(* CODESYS project Trabalho_final.project

Project tree, tasks and I/O mapping:
  Device : CODESYS Control Win V3, 3S - Smart Software Solutions GmbH, order no. 305021, version 3.5.11.40
    application Application
      libraries: Standard, * (System)
      task MainTask (cyclic, interval t#20ms, priority 1) calls Mode_Selection, Sequencia_Processo, Resetar, C_Automatico, Quantidade_Gin, Quantidade_Vermouth, Quantidade_tanque01, Quantidade_refrigerante, Temperatura, Quantidade_tanque02, c_resetar_tanque01, Sistema_esteira, C_Automatico_Tonel
      global variables GVL
      program Quantidade_Gin [ST]
      program Quantidade_Vermouth [ST]
      program Quantidade_refrigerante [ST]
      program Quantidade_tanque01 [ST]
      program Temperatura [ST]
      program C_Automatico [SFC]: Step3_active, Step7_active, Liga_motor_Abre_refrigerante_active, Resetar_active, Step3_active_0, Step2_active, Step4_active, Step5_active, Step6_active, Step7_active_0, Step8_active, Step10_active, Step9_active, Step12_active
      program Quantidade_tanque02 [ST]
      program Sistema_esteira [ST]
      program Mode_Selection [LD]
      program Resetar [ST]
      program Sequencia_Processo [SFC]: Step4_active, Automatico_active
      program c_resetar_tanque01 [ST]
      program C_Automatico_Tonel [SFC]: Step0_active, Step1_active, Step2_active, Step1_active_0
      program C_EMG [ST]
*)

// Device/Application/GVL
{attribute 'qualified_only'}
VAR_GLOBAL
	Mensagem : STRING[255] := 'NADA AINDA';
	
	//Modos de execução 
	Liga							  : BOOL;
	Sistema_ativo					  : BOOL;
	Selecao							  : BOOL := FALSE;  // 0 para automatico, 1 para o remoto
	Selecionado						  : BOOL;
	EMG								  : BOOL;	// Sistema de emergencia 
	Modo_manual 					  : BOOL;	// Indica que esta em modo manual
	Modo_automatico					  : BOOL;	// Indica que esta em modo automatico
	
	// controles do sistema 
	resetar : BOOL := FALSE;
	ativador_automatico	: BOOL := FALSE;
	resetar_tanque01 : BOOL := FALSE;
	
	// Colocar 30 litros de gin 
	Valvula_gin                       : BOOL := FALSE;   // Atuador válvula de gin
	Quantidade_gin					  : REAL := 0.0;     // Quantidade de gin (L)
	Temporizador_gin				  : TON; 			// De atuação 7,5S
	
	//Colocar 15 litros de vermouth 
	Valvula_vermouth                  : BOOL := FALSE;   // Válvula de vermouth
	Quantidade_vermouth			      : REAL := 0.0;     // Quantidade de vermouth (L)
	Temporizador_vermouth			  : TON;				// De atuação 4.5s 
	
	// Colocar Líquido Refrigerante
	Valvula_liquido_refrigerante      : BOOL := FALSE;   // Entrada de líquido refrigerante
	Quantidade_liquido_refrigerante	  : REAL := 0.0;     // Quantidade de liquido refrigerante (L)
	Valvula_descarte_refrigerante     : BOOL := FALSE;   // Válvula de descarte do refrigerante
    Alto_nivel_refrigerante           : BOOL := FALSE;   // Nível alto refrigerante
    Baixo_nivel_refrigerante          : BOOL := FALSE;   // Nível baixo refrigerante
	Temporizador_entrada_refrigerante : TON;
	Temporizador_saida_refrigerante : TON;
	
	// Tanque 01 quantidades 
	Tanque01_vazio                    : BOOL := TRUE;   // Sensor tanque 1 vazio
	Quantidade_liquido                : REAL := 0.0;     // Quantidade do líquido (L)
	Tanque01_30L                      : BOOL := FALSE;   // Sensor tanque(30L)
	Tanque01_45L                      : BOOL := FALSE;   // Sensor tanque(45L)
	Tanque01_50L                      : BOOL := FALSE;   // Sensor tanque(50L)
	Temporizador_produto			  : TON;
	Temporizador_produto_T2			  : TON;
	
	// Temperaturas
	Ativador_temperatura :BOOL:=FALSE;
 	Temporizador_temperatura		 : TON;
    Termometro_produto_0C            : BOOL := FALSE;   // Sensor que indica que a temperatura esta 0°c
	Temperatura_produto            	 : REAL := 27.0;     // Temperatura do produto
	
	//Bloco 01
	Motor_tanque01                   : BOOL := FALSE;   // Motor do tanque 01
	
	//Bloco de ligamento 
    Valvula_envio_produto            : BOOL := FALSE;   // Envio do produto
    Bomba_entre_tanques              : BOOL := FALSE;   // Bomba de transferência
    Valvula_rejeitos                 : BOOL := FALSE;   // Válvula para rejeitos
    Valvula_envio_tanque02           : BOOL := FALSE;   // Válvula de envio ao tanque 02
    
	//Bloco 02
	Tanque02_190l                    : BOOL := FALSE;   // Sensor tanque 2 cheio (190L)
	Quantidade_liquido_02            : REAL := 0.0;     // Quantidade do líquido em bloco 02 (L)
    Tanque02_95_por100               : BOOL := FALSE;   // Tanque 2 a 95% => 188,005 => 188L
    Tanque02_85_por100               : BOOL := FALSE;   // Tanque 2 a 85% => 168,215 => 168L
	Tanque02_50_por100               : BOOL := FALSE;   // Tanque 2 a 50% => 98,95 => 98L
    Tanque02_10_por100               : BOOL := FALSE;   // Tanque 2 a 10% => 19,79L  => 19L
	Temporizador_saida_tonel : TON;
	
	CarregamentoCompleto : BOOL:=FALSE;
	
	Timer_Inicia_Esvaziamento : TON;   // 5 segundos
    Timer_Retira_Produto : TON;       // 0.5 segundos
    Timer_Finaliza_Esgotamento : TON; // 3 segundos
	
	
	
	// Quantidade tonel 
    Valvula_produto_tonel            : BOOL := FALSE;   // Válvula para o tonel final
	Quantidade_liquido_tonel         : REAL := 0.0;     // Quantidade do líquido no tonel (L)
	Tonel_cheio                      : BOOL := FALSE;   // tonel cheio
	Tonel_pretaparado 				 : BOOL := FALSE;	// Sensor que indica que o tonel esta na boca da valvula
	Temporizador_produ_tonel		 : TON; 
	
	//Quantidade de toneis 
	Quantidade_tonel_produzido       : REAL := 0.0;     // Quantidade de toneis produzida
	Quantidade_tonel_liberada        : REAL := 0.0;     // Quantidade de toneis liberadas
	
	// esteira
    Esteira_tonel                    : BOOL := FALSE;   // Esteira transportadora
	Sensor_tonel 					 :BOOL := FALSE;
END_VAR

// Device/Application/Mode_Selection
PROGRAM Mode_Selection
VAR
END_VAR

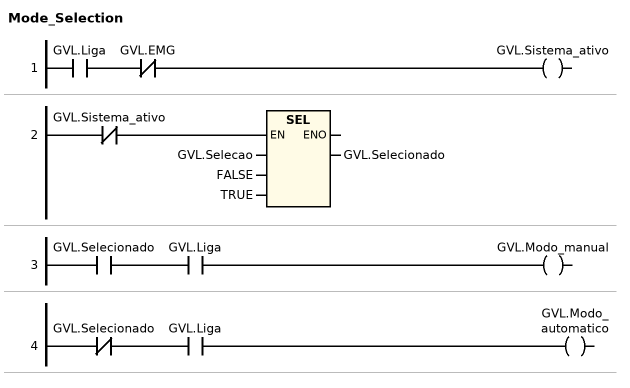
// NETWORK 1
GVL.Sistema_ativo := GVL.Liga AND NOT GVL.EMG;

// NETWORK 2
IF NOT GVL.Sistema_ativo THEN GVL.Selecionado := SEL(GVL.Selecao, FALSE, TRUE); END_IF

// NETWORK 3
GVL.Modo_manual := GVL.Selecionado AND GVL.Liga;

// NETWORK 4
GVL.Modo_automatico := NOT GVL.Selecionado AND GVL.Liga;

END_PROGRAM

// Device/Application/Sequencia_Processo
PROGRAM Sequencia_Processo
VAR
END_VAR

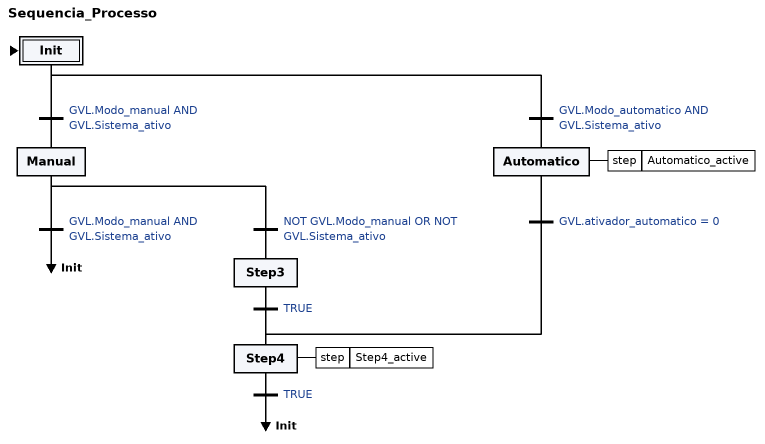
INITIAL_STEP Init:
END_STEP
TRANSITION FROM Init TO Manual
    := GVL.Modo_manual AND GVL.Sistema_ativo;
END_TRANSITION
STEP Manual:
END_STEP
TRANSITION FROM Manual TO Init
    := GVL.Modo_manual AND GVL.Sistema_ativo;
END_TRANSITION
TRANSITION FROM Manual TO Step3
    := NOT GVL.Modo_manual OR NOT GVL.Sistema_ativo;
END_TRANSITION
STEP Step3:
END_STEP
TRANSITION FROM Step3 TO Step4
    := TRUE;
END_TRANSITION
TRANSITION FROM Init TO Automatico
    := GVL.Modo_automatico AND GVL.Sistema_ativo;
END_TRANSITION
STEP Automatico:
    Automatico_active(N);  // step action
END_STEP
TRANSITION FROM Automatico TO Step4
    := GVL.ativador_automatico = 0;
END_TRANSITION
STEP Step4:
    Step4_active(N);  // step action
END_STEP
TRANSITION FROM Step4 TO Init
    := TRUE;
END_TRANSITION

ACTION Step4_active:
IF GVL.resetar = 0 THEN
	GVL.resetar := 1;
END_IF
END_ACTION

ACTION Automatico_active:
IF GVL.ativador_automatico = 0 THEN
	GVL.ativador_automatico := 1;
END_IF
END_ACTION

END_PROGRAM

// Device/Application/Resetar
PROGRAM Resetar
VAR
END_VAR


IF GVL.resetar = 1 THEN
	GVL.Valvula_gin                 			:= FALSE;
	GVL.Quantidade_gin              			:= 0.0;
	GVL.Valvula_vermouth            			:= FALSE;
	GVL.Quantidade_vermouth         			:= 0.0;
	GVL.Valvula_liquido_refrigerante 			:= FALSE;
	GVL.Quantidade_liquido_refrigerante			:= 0.0;
	GVL.Valvula_descarte_refrigerante 			:= FALSE;
	GVL.Alto_nivel_refrigerante      			:= FALSE;
	GVL.Baixo_nivel_refrigerante     			:= TRUE;
	GVL.Tanque01_vazio              			:= TRUE;
	GVL.Quantidade_liquido          			:= 0.0;
	GVL.Tanque01_30L                			:= FALSE;
	GVL.Tanque01_45L                			:= FALSE;
	GVL.Tanque01_50L                			:= FALSE;
	GVL.Termometro_produto_0C       			:= FALSE;
	GVL.Temperatura_produto         			:= 27.0;
	GVL.Motor_tanque01              			:= FALSE;
	GVL.Valvula_envio_produto       			:= FALSE;
	GVL.Bomba_entre_tanques         			:= FALSE;
	GVL.Valvula_rejeitos            			:= FALSE;
	GVL.Valvula_envio_tanque02      			:= FALSE;
	GVL.Tanque02_190l               			:= FALSE;
	GVL.Quantidade_liquido_02       			:= 0.0;
	GVL.Tanque02_95_por100          			:= FALSE;
	GVL.Tanque02_85_por100          			:= FALSE;
	GVL.Tanque02_50_por100          			:= FALSE;
	GVL.Tanque02_10_por100          			:= FALSE;
	GVL.Valvula_produto_tonel       			:= FALSE;
	GVL.Quantidade_liquido_tonel    			:= 0.0;
	GVL.Tonel_cheio                 			:= FALSE;
	GVL.Tonel_pretaparado           			:= FALSE;
	GVL.Quantidade_tonel_produzido  			:= 0.0;
	GVL.Quantidade_tonel_liberada   			:= 0.0;
	GVL.Esteira_tonel               			:= FALSE;
	GVL.resetar 								:= FALSE;
END_IF

END_PROGRAM

// Device/Application/Quantidade_Gin
PROGRAM Quantidade_Gin
VAR
	Limite_gin : REAL;
END_VAR

// ====================================================
//            CONTROLE DA VALVULA DE GIN
// ====================================================


// --------------------------------------
// Definição do limite por modo
// --------------------------------------
IF (GVL.Modo_manual = 1) THEN
    Limite_gin := 52;   // Modo Manual
ELSIF (GVL.Modo_automatico = 1) THEN
    Limite_gin := 30;   // Modo Automático
END_IF


// --------------------------------------
// Condições gerais de operação
// --------------------------------------
IF (GVL.EMG = 0) THEN

    // --------------------------------------
    // Se válvula está aberta
    // --------------------------------------
    IF GVL.Valvula_gin = 1 THEN

        // Fecha válvula quando atingir limite
        IF GVL.Quantidade_gin >= Limite_gin THEN
            GVL.Valvula_gin := 0;
        ELSE
            // Liga temporizador para contar 0.5 s
            GVL.Temporizador_gin(IN := TRUE, PT := T#0.5S);

            // Quando temporizador finalizar, incrementa volume
            IF GVL.Temporizador_gin.Q THEN

                //  equivalente a 4 L/s → 2 L a cada 0.5s
                GVL.Quantidade_gin      := GVL.Quantidade_gin + 2;
                GVL.Quantidade_liquido  := GVL.Quantidade_liquido + 2;

                // Reseta TON para permitir novo ciclo de 0.5s
                GVL.Temporizador_gin(IN := FALSE);
            END_IF

        END_IF

    ELSE
        // Válvula fechada → garantimos TON desligado
        GVL.Temporizador_gin(IN := FALSE);
    END_IF

ELSE
    // Se emergência ativa → TON off
    GVL.Temporizador_gin(IN := FALSE);
END_IF

END_PROGRAM

// Device/Application/Quantidade_Vermouth
PROGRAM Quantidade_Vermouth 
VAR
	Limite_vermouth : REAL;
END_VAR

// ====================================================
//        CONTROLE DA VÁLVULA DE VERMOUTH
// ====================================================


// --------------------------------------
// Definição do limite por modo
// --------------------------------------
IF (GVL.Modo_manual = 1) THEN
    Limite_vermouth := 51;    // Modo Manual → limite do líquido total
ELSIF (GVL.Modo_automatico = 1) THEN
    Limite_vermouth := 14;    // Modo Automático → limite específico do vermouth
END_IF



// --------------------------------------
// Condições gerais de operação
// --------------------------------------
IF (GVL.EMG = 0) THEN

    // --------------------------------------
    // Se a válvula está aberta
    // --------------------------------------
    IF GVL.Valvula_vermouth = 1 THEN

        // Fecha válvula quando atingir limite
        IF GVL.Quantidade_vermouth >= Limite_vermouth THEN

            GVL.Valvula_vermouth := 0;

            // Ajustes específicos do automático
            IF (GVL.Modo_automatico = 1) THEN
                GVL.Quantidade_liquido  := 45;
                GVL.Quantidade_vermouth := 15;
            END_IF

        ELSE
            // Liga temporizador para contar 0.5 s
            GVL.Temporizador_vermouth(IN := TRUE, PT := T#0.5S);

            // Quando temporizador finalizar, incrementa volume
            IF GVL.Temporizador_vermouth.Q THEN

                // Vazão: 3,33 L/s → 1,665 L a cada 0.5 s
                GVL.Quantidade_vermouth := GVL.Quantidade_vermouth + 1.665;
                GVL.Quantidade_liquido  := GVL.Quantidade_liquido  + 1.665;

                // Reseta TON para novo ciclo
                GVL.Temporizador_vermouth(IN := FALSE);
            END_IF

        END_IF

    ELSE
        // Válvula fechada → garante TON desligado
        GVL.Temporizador_vermouth(IN := FALSE);
    END_IF


ELSE
    // Se emergência ativa → TON desligado
    GVL.Temporizador_vermouth(IN := FALSE);
END_IF

END_PROGRAM

// Device/Application/C_Automatico
PROGRAM C_Automatico
VAR
END_VAR

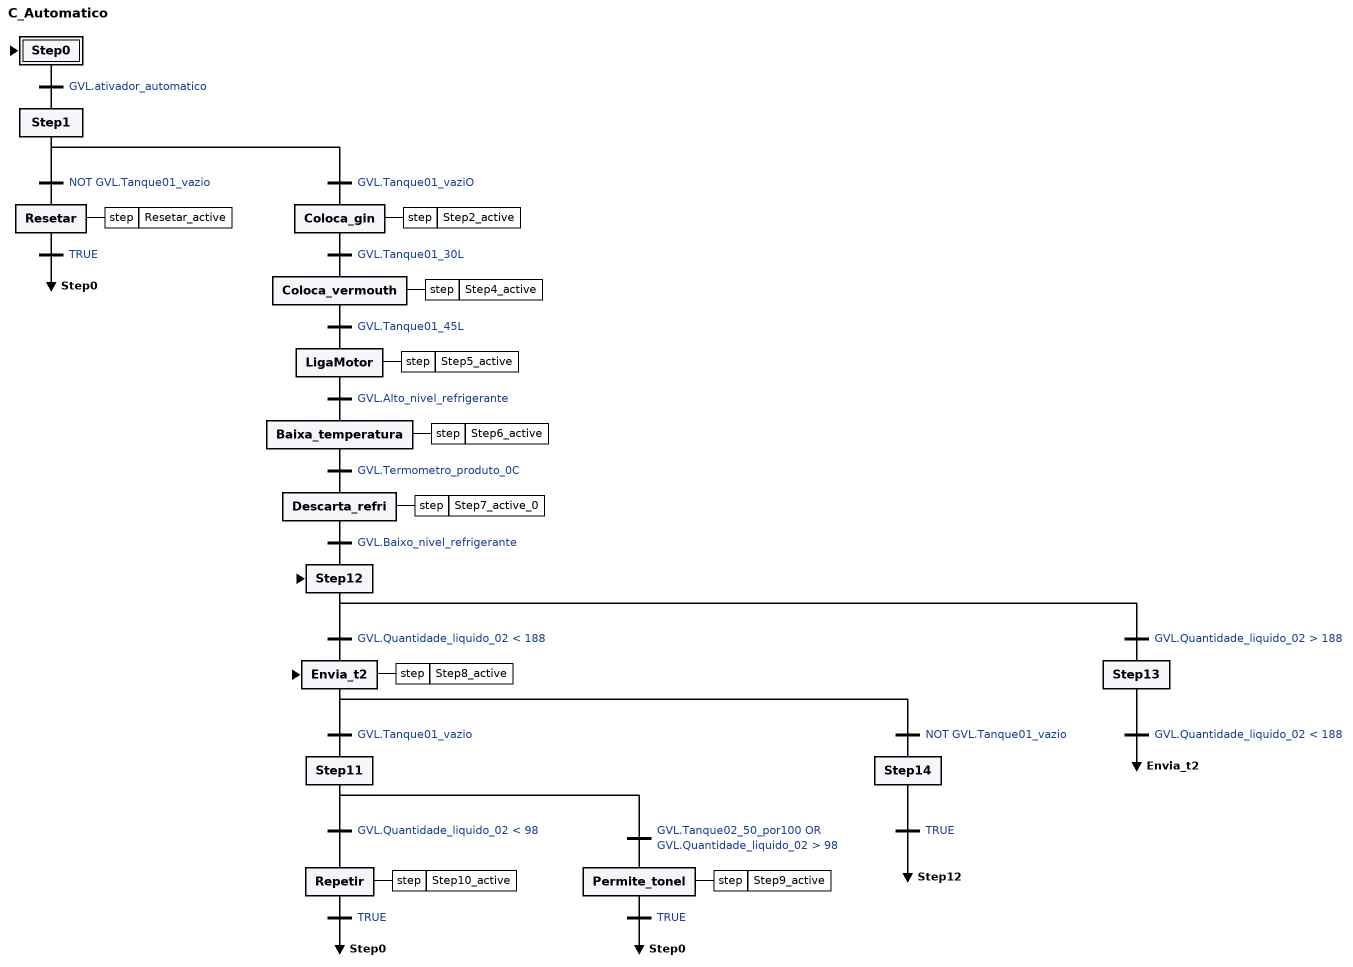
INITIAL_STEP Step0:
END_STEP
TRANSITION FROM Step0 TO Step1
    := GVL.ativador_automatico;
END_TRANSITION
STEP Step1:
END_STEP
TRANSITION FROM Step1 TO Resetar
    := NOT GVL.Tanque01_vazio;
END_TRANSITION
STEP Resetar:
    Resetar_active(N);  // step action
END_STEP
TRANSITION FROM Resetar TO Step0
    := TRUE;
END_TRANSITION
TRANSITION FROM Step1 TO Coloca_gin
    := GVL.Tanque01_vaziO;
END_TRANSITION
STEP Coloca_gin:
    Step2_active(N);  // step action
END_STEP
TRANSITION FROM Coloca_gin TO Coloca_vermouth
    := GVL.Tanque01_30L;
END_TRANSITION
STEP Coloca_vermouth:
    Step4_active(N);  // step action
END_STEP
TRANSITION FROM Coloca_vermouth TO LigaMotor
    := GVL.Tanque01_45L;
END_TRANSITION
STEP LigaMotor:
    Step5_active(N);  // step action
END_STEP
TRANSITION FROM LigaMotor TO Baixa_temperatura
    := GVL.Alto_nivel_refrigerante;
END_TRANSITION
STEP Baixa_temperatura:
    Step6_active(N);  // step action
END_STEP
TRANSITION FROM Baixa_temperatura TO Descarta_refri
    := GVL.Termometro_produto_0C;
END_TRANSITION
STEP Descarta_refri:
    Step7_active_0(N);  // step action
END_STEP
TRANSITION FROM Descarta_refri TO Step12
    := GVL.Baixo_nivel_refrigerante;
END_TRANSITION
STEP Step12:
END_STEP
TRANSITION FROM Step12 TO Envia_t2
    := GVL.Quantidade_liquido_02 < 188;
END_TRANSITION
TRANSITION FROM Step12 TO Step13
    := GVL.Quantidade_liquido_02 > 188;
END_TRANSITION
STEP Step13:
END_STEP
TRANSITION FROM Step13 TO Envia_t2
    := GVL.Quantidade_liquido_02 < 188;
END_TRANSITION
STEP Envia_t2:
    Step8_active(N);  // step action
END_STEP
TRANSITION FROM Envia_t2 TO Step11
    := GVL.Tanque01_vazio;
END_TRANSITION
TRANSITION FROM Envia_t2 TO Step14
    := NOT GVL.Tanque01_vazio;
END_TRANSITION
STEP Step14:
END_STEP
TRANSITION FROM Step14 TO Step12
    := TRUE;
END_TRANSITION
STEP Step11:
END_STEP
TRANSITION FROM Step11 TO Repetir
    := GVL.Quantidade_liquido_02 < 98;
END_TRANSITION
STEP Repetir:
    Step10_active(N);  // step action
END_STEP
TRANSITION FROM Repetir TO Step0
    := TRUE;
END_TRANSITION
TRANSITION FROM Step11 TO Permite_tonel
    := GVL.Tanque02_50_por100 OR GVL.Quantidade_liquido_02 > 98;
END_TRANSITION
STEP Permite_tonel:
    Step9_active(N);  // step action
END_STEP
TRANSITION FROM Permite_tonel TO Step0
    := TRUE;
END_TRANSITION

ACTION Step3_active:
GVL.Valvula_vermouth := 1;
END_ACTION

ACTION Step7_active:
GVL.Valvula_gin := 1;
END_ACTION

ACTION Liga_motor_Abre_refrigerante_active:
GVL.Valvula_liquido_refrigerante := 1;
GVL.Motor_tanque01 := 1;
END_ACTION

ACTION Resetar_active:
IF GVL.resetar = 0 THEN
	GVL.resetar := 1;
END_IF
END_ACTION

ACTION Step3_active_0:
GVL.ativador_automatico := FALSE;
END_ACTION

ACTION Step2_active:
GVL.Valvula_gin :=TRUE;
END_ACTION

ACTION Step4_active:
GVL.Valvula_vermouth := TRUE;
END_ACTION

ACTION Step5_active:
GVL.Motor_tanque01 := TRUE;
GVL.Valvula_liquido_refrigerante := TRUE;
END_ACTION

ACTION Step6_active:
IF (GVL.Quantidade_liquido_refrigerante = 15) AND (GVL.Motor_tanque01 = 1) AND (GVL.EMG = 0) THEN
	GVL.Ativador_temperatura := TRUE;
END_IF
END_ACTION

ACTION Step7_active_0:
GVL.Valvula_descarte_refrigerante:=TRUE;
END_ACTION

ACTION Step8_active:
GVL.Valvula_envio_produto := TRUE;
GVL.Bomba_entre_tanques := TRUE;
GVL.Valvula_envio_tanque02 := TRUE;
END_ACTION

ACTION Step10_active:
GVL.resetar_tanque01 := TRUE;
END_ACTION

ACTION Step9_active:
GVL.CarregamentoCompleto := True;
END_ACTION

ACTION Step12_active:
GVL.Tonel_cheio := FALSE;
GVL.Quantidade_liquido_tonel := 0;
GVL.Valvula_produto_tonel := TRUE;
END_ACTION

END_PROGRAM

// Device/Application/Quantidade_tanque01
PROGRAM Quantidade_tanque01
VAR
END_VAR

// =====================================================
//                 MODO MANUAL – ENVIO
// =====================================================

IF (GVL.Modo_manual = 1) AND (GVL.EMG = 0) THEN

    // Garante reset inicial
    GVL.Temporizador_produto(IN := FALSE);


    // -------------------------------------------------
    // ENVIO DE PRODUTO (válvula principal)
    // -------------------------------------------------
    IF (GVL.Valvula_envio_produto = 1) THEN

        // Só envia se bomba está ligada
        IF (GVL.Bomba_entre_tanques = 1) THEN

            // -------------------------------------------------
            // TANQUE 02 CHEIO → interrompe envio
            // -------------------------------------------------
            IF (GVL.Quantidade_liquido_02 >= 190)
               AND (GVL.Valvula_rejeitos = 0)
               AND (GVL.Valvula_envio_tanque02 = 1) THEN

                GVL.Valvula_envio_tanque02 := 0;
                GVL.Valvula_envio_produto  := 0;
                GVL.Bomba_entre_tanques    := 0;
            END_IF
			
			 IF (GVL.Quantidade_liquido > 0) THEN
				 // -------------------------------------------------
            	// ENVIO PARA TANQUE 02
            	// -------------------------------------------------
            	IF (GVL.Valvula_envio_tanque02 = 1) THEN
                
                	GVL.Temporizador_produto(IN := TRUE, PT := T#0.5S);

                	IF GVL.Temporizador_produto.Q THEN

                    	// 5 L para tanque 02
                    	GVL.Quantidade_liquido_02 := GVL.Quantidade_liquido_02 + 5;
                    	GVL.Quantidade_liquido    := GVL.Quantidade_liquido - 5;

                    	// Reset para novo ciclo
                    	GVL.Temporizador_produto(IN := FALSE);
                	END_IF


            	// -------------------------------------------------
            	// DESCARTE – quando tanque 02 não está recebendo
            	// -------------------------------------------------
            	ELSE
                	IF (GVL.Valvula_rejeitos = 1) THEN
                    
                    	GVL.Temporizador_produto(IN := TRUE, PT := T#0.5S);

                    	IF GVL.Temporizador_produto.Q THEN

                        	// 5 L descartados
                        	GVL.Quantidade_liquido := GVL.Quantidade_liquido - 5;

                        	GVL.Temporizador_produto(IN := FALSE);
                    	END_IF
                	END_IF
            	END_IF
			 ELSE
            	// Tanque vazio → desliga tudo
            	GVL.Valvula_envio_produto   := FALSE;
            	GVL.Valvula_rejeitos        := FALSE;
            	GVL.Valvula_envio_tanque02  := FALSE;
        	END_IF
        END_IF // bomba ligada
    ELSE
        // válvula de envio fechada → reset do TON
        GVL.Temporizador_produto(IN := FALSE);
    END_IF


    // -------------------------------------------------
    // INDICADORES DE NÍVEL DO TANQUE 01
    // -------------------------------------------------
    IF (GVL.Quantidade_liquido = 0) THEN
        GVL.Tanque01_vazio := 1;
        GVL.Tanque01_30L   := 0;
        GVL.Tanque01_45L   := 0;
        GVL.Tanque01_50L   := 0;
		
		// Reset de ingredientes
        GVL.Quantidade_gin       := 0;
        GVL.Quantidade_vermouth  := 0;

    ELSE
        GVL.Tanque01_vazio := 0;
        GVL.Tanque01_30L := (GVL.Quantidade_liquido = 30);
        GVL.Tanque01_45L := (GVL.Quantidade_liquido = 45);
        GVL.Tanque01_50L := (GVL.Quantidade_liquido = 50);
    END_IF

END_IF   // fim modo manual


// =====================================================
//             MODO AUTOMÁTICO – ENVIO
// =====================================================

IF (GVL.Modo_automatico = 1) AND (GVL.EMG = 0) THEN

    // -------------------------------------------------
    // ENVIO DE PRODUTO
    // -------------------------------------------------
    IF (GVL.Valvula_envio_produto = 1) THEN

        // Tanque com volume > 0
        IF (GVL.Quantidade_liquido > 0) THEN

			// -------------------------------------------------
            // TANQUE 02 CHEIO → interrompe envio
            // -------------------------------------------------
            IF (GVL.Quantidade_liquido_02 >= 190)
               AND (GVL.Valvula_rejeitos = 0)
               AND (GVL.Valvula_envio_tanque02 = 1) THEN

                GVL.Valvula_envio_tanque02 := 0;
                GVL.Valvula_envio_produto  := 0;
                GVL.Bomba_entre_tanques    := 0;
            END_IF
			
            // ---------------------------
            // ENVIO PARA TANQUE 02
            // ---------------------------
            IF (GVL.Valvula_envio_tanque02 = 1) THEN

                GVL.Temporizador_produto_T2(IN := TRUE, PT := T#0.5S);

                IF (GVL.Temporizador_produto_T2.Q) THEN

                    GVL.Quantidade_liquido_02 := GVL.Quantidade_liquido_02 + 5;
                    GVL.Quantidade_liquido    := GVL.Quantidade_liquido - 5;

                    GVL.Temporizador_produto_T2(IN := FALSE);
                END_IF
            END_IF

            // ---------------------------
            // DESCARTE
            // ---------------------------
            IF (GVL.Valvula_rejeitos = 1) THEN

                GVL.Temporizador_produto(IN := TRUE, PT := T#0.5S);

                IF (GVL.Temporizador_produto.Q) THEN

                    GVL.Quantidade_liquido := GVL.Quantidade_liquido - 5;

                    GVL.Temporizador_produto(IN := FALSE);
                END_IF
            END_IF

        ELSE
            // Tanque vazio → desliga tudo
            GVL.Valvula_envio_produto   := FALSE;
            GVL.Valvula_rejeitos        := FALSE;
            GVL.Valvula_envio_tanque02  := FALSE;
        END_IF
    END_IF


    // -------------------------------------------------
    // INDICADORES DE NÍVEL DO TANQUE 01
    // -------------------------------------------------
    IF (GVL.Quantidade_liquido = 0) THEN
        GVL.Tanque01_vazio := 1;
        GVL.Tanque01_30L   := 0;
        GVL.Tanque01_45L   := 0;
        GVL.Tanque01_50L   := 0;

        // Reset de ingredientes
        GVL.Quantidade_gin       := 0;
        GVL.Quantidade_vermouth  := 0;

    ELSE
        GVL.Tanque01_vazio := 0;

        GVL.Tanque01_30L := (GVL.Quantidade_liquido = 30);
        GVL.Tanque01_45L := (GVL.Quantidade_liquido = 45);
        GVL.Tanque01_50L := (GVL.Quantidade_liquido = 50);
    END_IF

END_IF   // fim modo automático

END_PROGRAM

// Device/Application/Quantidade_refrigerante
PROGRAM Quantidade_refrigerante
VAR
	Limite_entrada: REAL;
END_VAR

(* =====================================================
                 CONTROLE – ENTRADA
   ===================================================== *)

(* --------------------------------------
   Definição do limite por modo
   -------------------------------------- *)
IF (GVL.Modo_manual = 1) THEN
    Limite_entrada := 15;        (* Manual *)
ELSIF (GVL.Modo_automatico = 1) THEN
    Limite_entrada := 15;        (* Automático *)
END_IF;


(* --------------------------------------
   Condições gerais de operação
   -------------------------------------- *)
IF (GVL.EMG = 0) THEN

    (* Válvula aberta *)
    IF (GVL.Valvula_liquido_refrigerante = 1) THEN

        (* Já atingiu o limite *)
        IF (GVL.Quantidade_liquido_refrigerante >= Limite_entrada) THEN

            GVL.Valvula_liquido_refrigerante := 0;
            GVL.Quantidade_liquido_refrigerante := Limite_entrada;

            GVL.Alto_nivel_refrigerante  := 1;
            GVL.Baixo_nivel_refrigerante := 0;

        ELSE
            (* Nível ainda baixo *)
            GVL.Alto_nivel_refrigerante  := 0;
            GVL.Baixo_nivel_refrigerante := 1;

            (* Temporizador de 0.5s *)
            GVL.Temporizador_entrada_refrigerante(IN := TRUE, PT := T#0.5S);

            IF GVL.Temporizador_entrada_refrigerante.Q THEN

                (* Incremento 1.665 L a cada 0.5s *)
                GVL.Quantidade_liquido_refrigerante :=
                    GVL.Quantidade_liquido_refrigerante + 1.665;

                (* Reset do TON *)
                GVL.Temporizador_entrada_refrigerante(IN := FALSE);
            END_IF
        END_IF

    ELSE
        (* Válvula fechada → TON desligado *)
        GVL.Temporizador_entrada_refrigerante(IN := FALSE);
    END_IF

ELSE
    (* Emergência → força TON desligado *)
    GVL.Temporizador_entrada_refrigerante(IN := FALSE);
END_IF;


(* =====================================================
                 CONTROLE – SAÍDA
   ===================================================== *)

(* Sem limite → descarrega até chegar a zero *)

IF (GVL.EMG = 0) THEN

    IF (GVL.Valvula_descarte_refrigerante = 1) THEN

        (* Se já está vazio *)
        IF (GVL.Quantidade_liquido_refrigerante <= 0) THEN
            
            GVL.Valvula_descarte_refrigerante := 0;
            GVL.Quantidade_liquido_refrigerante := 0;

            GVL.Alto_nivel_refrigerante  := 0;
            GVL.Baixo_nivel_refrigerante := 1;

        ELSE
            (* Ainda há líquido para descarregar *)
            GVL.Alto_nivel_refrigerante  := 1;
            GVL.Baixo_nivel_refrigerante := 0;

            (* Temporizador 0.5s *)
            GVL.Temporizador_saida_refrigerante(IN := TRUE, PT := T#0.5S);

            IF GVL.Temporizador_saida_refrigerante.Q THEN

                (* Decremento 1.665 L a cada 0.5s *)
                GVL.Quantidade_liquido_refrigerante :=
                    GVL.Quantidade_liquido_refrigerante - 1.665;

                (* Reset TON *)
                GVL.Temporizador_saida_refrigerante(IN := FALSE);
            END_IF

        END_IF

    ELSE
        GVL.Temporizador_saida_refrigerante(IN := FALSE);
    END_IF

ELSE
    (* Emergência *)
    GVL.Temporizador_saida_refrigerante(IN := FALSE);
END_IF;

END_PROGRAM

// Device/Application/Temperatura
PROGRAM Temperatura
VAR
END_VAR

// =====================================================
//              RESFRIAMENTO DO PRODUTO
// =====================================================

// O bloco só atua se o ativador estiver ligado
IF (GVL.Ativador_temperatura = TRUE) THEN

    // ----------------------------------------------
    // Enquanto temperatura maior que 0°C → resfriar
    // ----------------------------------------------
    IF (GVL.Temperatura_produto > 0) THEN

        // TON de 1 segundo
        GVL.Temporizador_temperatura(IN := TRUE, PT := T#1S);

        // Quando completar 1 segundo → reduz 1°C
        IF (GVL.Temporizador_temperatura.Q) THEN

            // Evita temperatura negativa
            IF (GVL.Temperatura_produto > 0) THEN
                GVL.Temperatura_produto := GVL.Temperatura_produto - 1;
            END_IF

            // Reset do TON para novo ciclo
            GVL.Temporizador_temperatura(IN := FALSE);
        END_IF

    // ----------------------------------------------
    // Quando chegar a 0°C → finaliza operação
    // ----------------------------------------------
    ELSE
        // Garante temperatura mínima
        GVL.Temperatura_produto := 0;

        // Desativa processo
        GVL.Ativador_temperatura := FALSE;

        // Ativa indicador de temperatura final
        GVL.Termometro_produto_0C := 1;

        // Desliga motor do tanque
        GVL.Motor_tanque01 := 0;

        // Segurança: desliga TON
        GVL.Temporizador_temperatura(IN := FALSE);

    END_IF

END_IF;

END_PROGRAM

// Device/Application/Quantidade_tanque02
PROGRAM Quantidade_tanque02
VAR
END_VAR

// =====================================================
//      CONTROLE DE TRANSFERÊNCIA PARA O TONEL
// =====================================================


// =====================================================
//                  MODO MANUAL
// =====================================================

IF (GVL.Modo_manual = 1) AND (GVL.EMG = 0) THEN

    // --------------------------------------
    // Válvula aberta → inicia transferência
    // --------------------------------------
    IF (GVL.Valvula_produto_tonel = 1) THEN
		
		IF GVL.Quantidade_liquido_02 > 1 THEN
			// Liga TON com período de 0.5s
        	GVL.Temporizador_saida_tonel(IN := TRUE, PT := T#0.5S);

        	// Quando o TON completar o ciclo
        	IF (GVL.Temporizador_saida_tonel.Q) THEN

            	IF GVL.Tonel_pretaparado THEN
					// Verifica limite para NÃO ultrapassar 15 L no tonel
            		IF (GVL.Quantidade_liquido_tonel < 15) THEN
                		// 1 L por ciclo de 0.5s
                		GVL.Quantidade_liquido_02 := GVL.Quantidade_liquido_02 - 1;
                		GVL.Quantidade_liquido_tonel := GVL.Quantidade_liquido_tonel + 1;
            		ELSE
                		// Tonel cheio → fecha válvula
                		GVL.Valvula_produto_tonel := 0;
            		END_IF
				ELSE
					GVL.Quantidade_liquido_02 := GVL.Quantidade_liquido_02 - 1;
				END_IF

            	// Reseta TON para um novo ciclo
            	GVL.Temporizador_saida_tonel(IN := FALSE);
        	END_IF
		END_IF

    ELSE
        // Válvula fechada → desliga TON
        GVL.Temporizador_saida_tonel(IN := FALSE);
    END_IF

END_IF



// =====================================================
//                 MODO AUTOMÁTICO
// =====================================================

IF (GVL.Modo_automatico = 1) AND (GVL.EMG = 0) THEN

    // --------------------------------------
    // Só funciona se tonel não está cheio
    // --------------------------------------
    IF (GVL.Valvula_produto_tonel = 1) AND (GVL.Tonel_cheio = 0) THEN
		IF GVL.Quantidade_liquido_02 > 1 AND GVL.Tonel_pretaparado  THEN
			// Se ainda cabe líquido no tonel
        	IF (GVL.Quantidade_liquido_tonel < 15) THEN
            	// Liga TON de 0.5s
            	GVL.Temporizador_saida_tonel(IN := TRUE, PT := T#0.5S);
				
            	IF (GVL.Temporizador_saida_tonel.Q) THEN

                	// Transferência 1 L por ciclo
                	GVL.Quantidade_liquido_02 := GVL.Quantidade_liquido_02 - 1;
                	GVL.Quantidade_liquido_tonel := GVL.Quantidade_liquido_tonel + 1;

                	// Reseta TON
                	GVL.Temporizador_saida_tonel(IN := FALSE);
            	END_IF

        	ELSE
            	// Tonel está cheio → válvula fecha
            	GVL.Valvula_produto_tonel := 0;
        	END_IF
		ELSE
			GVL.Valvula_produto_tonel := FALSE;
		END_IF
    ELSE
        // Se tonel está cheio ou válvula fechada → garante fechamento
        GVL.Valvula_produto_tonel := 0;
        GVL.Temporizador_saida_tonel(IN := FALSE);
    END_IF

END_IF



// =====================================================
//      SINALIZAÇÃO DE NÍVEIS DO TANQUE 02
// =====================================================

// ---- 95% ----
IF (GVL.Quantidade_liquido_02 = 188) THEN
    GVL.Tanque02_95_por100 := 1;
    GVL.Tanque02_85_por100 := 0;
    GVL.Tanque02_50_por100 := 0;
    GVL.Tanque02_10_por100 := 0;
	GVL.CarregamentoCompleto := TRUE;
END_IF

// ---- 85% ----
IF (GVL.Quantidade_liquido_02 = 168) THEN
    GVL.Tanque02_95_por100 := 0;
    GVL.Tanque02_85_por100 := 1;
    GVL.Tanque02_50_por100 := 0;
    GVL.Tanque02_10_por100 := 0;
	GVL.CarregamentoCompleto := TRUE;
END_IF

// ---- 50% ----
IF (GVL.Quantidade_liquido_02 = 98) THEN
    GVL.Tanque02_95_por100 := 0;
    GVL.Tanque02_85_por100 := 0;
    GVL.Tanque02_50_por100 := 1;
    GVL.Tanque02_10_por100 := 0;
	GVL.CarregamentoCompleto := TRUE;
    GVL.Esteira_tonel := 1;
END_IF

// ---- 10% ----
IF (GVL.Quantidade_liquido_02 = 19) THEN
    GVL.Tanque02_95_por100 := 0;
    GVL.Tanque02_85_por100 := 0;
    GVL.Tanque02_50_por100 := 0;
    GVL.Tanque02_10_por100 := 1;
    GVL.CarregamentoCompleto := FALSE;
END_IF

END_PROGRAM

// Device/Application/c_resetar_tanque01
PROGRAM c_resetar_tanque01
VAR
END_VAR

IF GVL.resetar_tanque01 THEN
	GVL.Valvula_gin := FALSE;
	GVL.Quantidade_gin := 0;
	GVL.Valvula_vermouth := FALSE;
	GVL.Quantidade_vermouth := 0;
	GVL.Valvula_liquido_refrigerante := FALSE;
	GVL.Quantidade_liquido_refrigerante := 0;
	GVL.Valvula_descarte_refrigerante := FALSE;
	GVL.Quantidade_liquido := 0;
	GVL.Ativador_temperatura := FALSE;
	GVL.Termometro_produto_0C := FALSE;
	GVL.Temperatura_produto :=27;
	GVL.Motor_tanque01 := FALSE;
	GVL.Valvula_envio_produto := FALSE;
	GVL.Bomba_entre_tanques := FALSE;
	GVL.Valvula_rejeitos := FALSE;
	GVL.Valvula_envio_tanque02 := FALSE;
	GVL.resetar_tanque01 := FALSE;
END_IF

END_PROGRAM

// Device/Application/Sistema_esteira
PROGRAM Sistema_esteira
VAR
END_VAR

IF (GVL.Modo_automatico = 1) AND (GVL.EMG = 0) THEN
    
    // ============================
    // PRODUÇÃO DE TONÉIS
    // ============================
    
    // Se a esteira está ligada e ainda não atingiu 3 tonéis
    IF (GVL.Esteira_tonel = TRUE) AND (GVL.Quantidade_tonel_produzido < 3) THEN
        
        // Inicia TON de 15s
        GVL.Temporizador_produ_tonel(IN := TRUE, PT := T#15S);

        // Quando o TON completar 15s → produz 1 tonel
        IF GVL.Temporizador_produ_tonel.Q THEN
            GVL.Quantidade_tonel_produzido := GVL.Quantidade_tonel_produzido + 1;
            GVL.Temporizador_produ_tonel(IN := FALSE);    // reset do timer
        END_IF

    ELSE
        // Caso já tenha produzido 3 tonéis → para a esteira
        GVL.Esteira_tonel := FALSE;
        GVL.Tonel_pretaparado := TRUE;

        // Garante que o timer não fique rodando
        GVL.Temporizador_produ_tonel(IN := FALSE);
    END_IF

END_IF


// Logica para computar toneis produzidos 
IF GVL.Modo_automatico = 1 AND GVL.EMG = 0 THEN
	IF GVL.Tonel_cheio THEN
		GVL.Quantidade_tonel_liberada := GVL.Quantidade_tonel_liberada + 1;
		GVL.Quantidade_tonel_produzido := GVL.Quantidade_tonel_produzido - 1;
		GVL.Quantidade_liquido_tonel := 0;
		GVL.Tonel_cheio := FALSE;
	END_IF
END_IF

END_PROGRAM

// Device/Application/C_Automatico_Tonel
PROGRAM C_Automatico_Tonel
VAR
END_VAR

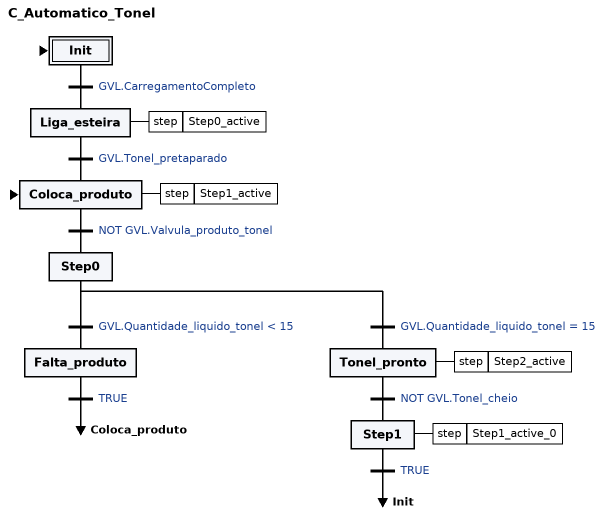
INITIAL_STEP Init:
END_STEP
TRANSITION FROM Init TO Liga_esteira
    := GVL.CarregamentoCompleto;
END_TRANSITION
STEP Liga_esteira:
    Step0_active(N);  // step action
END_STEP
TRANSITION FROM Liga_esteira TO Coloca_produto
    := GVL.Tonel_pretaparado;
END_TRANSITION
STEP Coloca_produto:
    Step1_active(N);  // step action
END_STEP
TRANSITION FROM Coloca_produto TO Step0
    := NOT GVL.Valvula_produto_tonel;
END_TRANSITION
STEP Step0:
END_STEP
TRANSITION FROM Step0 TO Falta_produto
    := GVL.Quantidade_liquido_tonel < 15;
END_TRANSITION
STEP Falta_produto:
END_STEP
TRANSITION FROM Falta_produto TO Coloca_produto
    := TRUE;
END_TRANSITION
TRANSITION FROM Step0 TO Tonel_pronto
    := GVL.Quantidade_liquido_tonel = 15;
END_TRANSITION
STEP Tonel_pronto:
    Step2_active(N);  // step action
END_STEP
TRANSITION FROM Tonel_pronto TO Step1
    := NOT GVL.Tonel_cheio;
END_TRANSITION
STEP Step1:
    Step1_active_0(N);  // step action
END_STEP
TRANSITION FROM Step1 TO Init
    := TRUE;
END_TRANSITION

ACTION Step0_active:
GVL.Esteira_tonel := 1;
END_ACTION

ACTION Step1_active:
GVL.Valvula_produto_tonel := 1;
END_ACTION

ACTION Step2_active:
GVL.Tonel_cheio := TRUE;
GVL.Tonel_pretaparado := FALSE;
END_ACTION

ACTION Step1_active_0:
IF GVL.Quantidade_liquido_02 >= 98 THEN
	GVL.CarregamentoCompleto := TRUE;
ELSE
	GVL.CarregamentoCompleto := FALSE;
END_IF
END_ACTION

END_PROGRAM

// Device/Application/C_EMG
PROGRAM C_EMG
VAR
END_VAR

// =======================================
//         TRATAMENTO DE EMERGÊNCIA
// =======================================

IF GVL.EMG THEN

    // ---------------------------
    // 1) FECHAR VÁLVULAS IMEDIATAMENTE
    // ---------------------------
    GVL.Valvula_gin := FALSE;
    GVL.Valvula_vermouth := FALSE;
    GVL.Valvula_liquido_refrigerante := FALSE;

    // Ativa timer de 5s para iniciar o esvaziamento
    GVL.Timer_Inicia_Esvaziamento(IN := TRUE, PT := T#5S);

    // ---------------------------
    // 2) APÓS 5s — COMEÇA O ESVAZIAMENTO
    // ---------------------------
    IF GVL.Timer_Inicia_Esvaziamento.Q THEN
        
        // Liga bomba e válvula de rejeito
        GVL.Bomba_entre_tanques := TRUE;
        GVL.Valvula_rejeitos := TRUE;

        // Temporizador de remoção (0.5s)
        GVL.Timer_Retira_Produto(IN := TRUE, PT := T#0.5S);

        // A cada 0.5 segundos, remove 5 unidades
        IF GVL.Timer_Retira_Produto.Q THEN
            IF GVL.Quantidade_liquido > 0 THEN
                GVL.Quantidade_liquido := GVL.Quantidade_liquido - 5;
            END_IF;
            
            GVL.Timer_Retira_Produto(IN := FALSE); // reset
        END_IF

        // -------------------------------
        // 3) QUANDO O TANQUE ZERAR
        // -------------------------------
        IF GVL.Quantidade_liquido <= 0 THEN
            
            // Desliga o timer de retirada
            GVL.Timer_Retira_Produto(IN := FALSE);

            // Inicia timer de 3 segundos pós-esvaziamento
            GVL.Timer_Finaliza_Esgotamento(IN := TRUE, PT := T#3S);

            // -------------------------------
            // 4) APÓS OS 3 SEGUNDOS FINAIS
            // -------------------------------
            IF GVL.Timer_Finaliza_Esgotamento.Q THEN
                
                GVL.Valvula_rejeitos := FALSE;
                GVL.Bomba_entre_tanques := FALSE;

                // ---------------------------
                // 5) ENCERRA SISTEMA E EMG
                // ---------------------------
                GVL.Liga := FALSE;
                GVL.EMG := FALSE;

                // Reset de timers
                GVL.Timer_Inicia_Esvaziamento(IN := FALSE);
                GVL.Timer_Finaliza_Esgotamento(IN := FALSE);
            END_IF
        END_IF
    END_IF
END_IF

END_PROGRAM
